Yaskawa INFORM job: R1_W49-52-A1(90,180)KM-OK.JBI

/JOB
//NAME R1_W49-52-A1(90,180)KM-OK
///FOLDERNAME KRIS-SCIANA
//POS
///NPOS 81,81,0,5,0,0
///TOOL 0
///POSTYPE PULSE
///PULSE
C00000=-7587,-78695,-93296,1458,74884,57665
C00001=105558,-78695,-93296,1458,74884,57665
C00002=105558,-78695,-93296,1458,74884,57665
C00003=54740,-7974,-10006,12021,87689,28506
C00004=74776,32390,22089,16092,92623,17270
C00005=74867,35757,29537,16050,89859,16941
C00006=75036,36599,32361,16047,88568,16832
C00007=75036,36895,33395,16047,88102,16772
C00008=74903,37254,32698,16044,88719,16805
C00009=72459,12362,8558,16008,91190,16266
C00010=61209,-17232,-1681,36622,66784,6421
C00011=61731,-16191,-908,36534,66611,6591
C00012=59990,-21702,-9204,36261,69196,6738
C00013=72720,3761,1433,15340,81732,21663
C00014=72610,7758,8804,15444,79356,21325
C00015=73045,10828,13692,15468,77892,21294
C00016=73045,11312,15266,15506,77198,21205
C00017=73045,10828,13692,15468,77892,21294
C00018=73056,12709,16349,15503,77245,21214
C00019=72823,14370,17858,15529,77218,21128
C00020=73056,12283,14967,15470,77854,21292
C00021=79642,10121,9779,4752,79820,25647
C00022=80358,6534,2777,4651,82236,25983
C00023=69953,-20577,-2415,29105,71989,-2082
C00024=71388,-15105,4995,29275,69960,-2047
C00025=71943,-12839,8075,29360,69127,-2048
C00026=71949,-11985,10076,29503,68430,-2234
C00027=71943,-12839,8075,29360,69127,-2048
C00028=78156,-21778,1298,21120,59983,2481
C00029=78744,-20042,2543,20963,59953,2712
C00030=78156,-21778,1298,21120,59983,2481
C00031=77865,-24315,-1842,21059,60645,2495
C00032=77104,-30529,-9436,20946,62223,2499
C00033=66753,-24791,-5212,33273,69818,-4262
C00034=68453,-19258,1867,33429,67885,-4157
C00035=68354,-14056,6987,33541,67521,-4315
C00036=68354,-13519,8242,33651,67105,-4449
C00037=68354,-12784,9926,33801,66552,-4629
C00038=68354,-12923,9607,33773,66657,-4594
C00039=69108,-16977,4805,33509,67096,-4131
C00040=78682,-30038,-3543,25118,55124,1302
C00041=79303,-28327,-2398,24897,55100,1566
C00042=78682,-30038,-3543,25118,55124,1302
C00043=75986,-28450,-4438,25449,57169,654
C00044=75599,-31023,-7408,25413,57744,634
C00045=74583,-37366,-14608,25368,59113,542
C00046=54832,-34796,3895,72693,39731,39244
C00047=56965,-32089,5608,72268,38461,39820
C00048=57588,-30877,10011,80435,36175,35219
C00049=57943,-31847,4343,71137,38137,40613
C00050=56828,-32279,5486,72299,38543,39782
C00051=56257,-29828,13363,87123,37301,31673
C00052=56951,-32108,5596,72272,38470,39816
C00053=54817,-34814,3883,72695,39739,39240
C00054=70512,18761,16215,24928,63616,33333
C00055=71552,23284,21050,24721,62713,33555
C00056=71200,18616,16875,24804,62971,33467
C00057=70825,17807,14425,24705,64080,33568
C00058=67755,12532,11412,25844,64241,32344
C00059=67541,9161,7476,25769,64930,32423
C00060=66799,6994,5573,25983,65214,32188
C00061=71450,3986,10861,16686,71001,58886
C00062=83506,38901,46150,14860,73867,63488
C00063=83544,40808,50439,14978,72254,63301
C00064=72489,19688,28494,17099,68495,-19316
C00065=72729,20279,28486,17025,68740,-19190
C00066=86246,35765,44483,7660,69456,64556
C00067=83439,39894,48722,4111,67251,63742
C00068=81920,28066,37949,6469,61442,62824
C00069=80051,2111,23117,10924,39735,59719
C00070=82415,-8846,23843,4944,20359,59825
C00071=68873,-12309,21104,25070,22681,48537
C00072=68288,-12793,20764,25848,22814,48089
C00073=68024,-12940,20839,26306,22782,47835
C00074=67958,-13479,20947,26756,22492,47608
C00075=67911,-23908,2369,21552,28082,50172
C00076=67911,-23908,2369,21552,28082,50172
C00077=73405,-104993,-53637,20388,20000,51360
C00078=27978,-168994,-134866,21563,-5876,50681
C00079=117827,-168994,-134866,21563,-5876,50681
C00080=64827,-168994,-134866,21563,-5876,50681
BC00000=61902,753087,991662
BC00001=7382,751982,991662
BC00002=7382,1232959,991662
BC00003=41401,1216769,518914
BC00004=54510,1210531,336745
BC00005=54510,1189341,336745
BC00006=54510,1189341,336745
BC00007=54510,1189341,336745
BC00008=54510,1189341,336745
BC00009=54510,1189341,336745
BC00010=54510,1189341,336745
BC00011=54510,1189341,336745
BC00012=54510,1189341,336745
BC00013=82383,1191142,368989
BC00014=82383,1191142,368989
BC00015=82383,1191142,368989
BC00016=82383,1191142,368989
BC00017=82383,1191142,368989
BC00018=82383,1191142,368989
BC00019=82383,1191142,368989
BC00020=82383,1191142,368989
BC00021=82383,1191142,368989
BC00022=82383,1191142,368989
BC00023=120081,1191142,413938
BC00024=120081,1191142,413938
BC00025=120081,1191142,413938
BC00026=120081,1191142,413938
BC00027=120081,1191142,413938
BC00028=120081,1191142,413938
BC00029=120081,1191142,413938
BC00030=120081,1191142,413938
BC00031=120081,1191142,413938
BC00032=120081,1191142,413938
BC00033=92240,1191142,398030
BC00034=92240,1191142,398030
BC00035=92240,1191142,398030
BC00036=92240,1191142,398030
BC00037=92240,1191142,398030
BC00038=92240,1191142,398030
BC00039=92240,1191142,398030
BC00040=92240,1191142,398030
BC00041=92240,1191142,398030
BC00042=92240,1191142,398030
BC00043=92240,1191142,398030
BC00044=92240,1191142,398030
BC00045=92240,1191142,398030
BC00046=53400,1191142,369839
BC00047=54054,1191142,349350
BC00048=54316,1191142,341155
BC00049=54316,1191142,341155
BC00050=54316,1191142,341155
BC00051=86854,1191142,340272
BC00052=86592,1191142,348467
BC00053=85937,1191142,368955
BC00054=29761,1191142,318980
BC00055=30700,1191142,309584
BC00056=30700,1191142,309584
BC00057=30700,1191142,309584
BC00058=37841,1191142,292738
BC00059=36902,1191142,302135
BC00060=34556,1191142,325626
BC00061=58988,1191142,416009
BC00062=58988,1191142,416009
BC00063=58988,1191142,416009
BC00064=57963,1191142,388162
BC00065=57963,1191142,388162
BC00066=58988,1191142,416009
BC00067=58988,1191142,416009
BC00068=58988,1191142,416009
BC00069=58988,1191142,416009
BC00070=58988,1191142,416008
BC00071=58988,1191142,416008
BC00072=58988,1191142,416008
BC00073=58988,1191142,416008
BC00074=58988,1191142,416008
BC00075=58988,1191142,416008
BC00076=58988,1191142,416008
BC00077=58988,1191142,416008
BC00078=8928,1190598,1065226
BC00079=8928,1190598,1065226
BC00080=8928,698634,1065226
///POSTYPE BASE
///RECTAN
///RCONF 0,0,0,0,0,0,0,0,0,0,0,0,0,0,0,0,0,0,0,0,0,0,0,0
P00006=0.222,-3.123,-1.508,0.0000,0.0000,0.0000
P00023=0.143,-0.036,0.682,0.0000,0.0000,0.0000
P00024=0.145,-0.552,1.326,0.0000,0.0000,0.0000
P00026=0.562,-0.002,-0.337,0.0000,0.0000,0.0000
P00027=-0.746,0.015,-9.096,0.0000,0.0000,0.0000
//INST
///DATE 2024/07/25 10:26
///ATTR SC,RW
///GROUP1 RB1,BS1
NOP
'r1_W49-52-A1(90,180)
SFTOF
MOVJ C00000 BC00000 VJ=80.00
MOVJ C00001 BC00001 VJ=80.00
MOVJ C00002 BC00002 VJ=80.00
MOVJ C00003 BC00003 VJ=100.00
MOVJ C00004 BC00004 VJ=50.00
MOVJ C00005 BC00005 VJ=20.00
MOVL C00006 BC00006 V=60.0
REFP 3 C00007 BC00007
CALL JOB:SEARCH-R1
SET P026 P006
SFTON P026
MOVL C00008 BC00008 V=60.0
MOVL C00009 BC00009 V=100.0
MOVL C00010 BC00010 V=83.3
REFP 3 C00011 BC00011
CALL JOB:SEARCH-R1
SET P026 P006
SFTON P026
MOVL C00012 BC00012 V=60.0
'Path S1206
SFTOF
MOVJ C00013 BC00013 VJ=50.00
MOVJ C00014 BC00014 VJ=50.00
MOVL C00015 BC00015 V=60.0
REFP 3 C00016 BC00016
CALL JOB:SEARCH-R1
SET P024 P006
SFTON P024
MOVL C00017 BC00017 V=100.0
MOVL C00018 BC00018 V=60.0
REFP 3 C00019 BC00019
CALL JOB:SEARCH-R1
SET P024 P006
SFTON P024
MOVL C00020 BC00020 V=60.0
MOVL C00021 BC00021 V=100.0
MOVL C00022 BC00022 V=166.7
'Path S1207
SFTOF
MOVJ C00023 BC00023 VJ=50.00
MOVJ C00024 BC00024 VJ=50.00
MOVL C00025 BC00025 V=133.3
REFP 3 C00026 BC00026
CALL JOB:SEARCH-R1
SET P023 P006
SFTON P023
MOVL C00027 BC00027 V=60.0
MOVL C00028 BC00028 V=60.0
REFP 3 C00029 BC00029
CALL JOB:SEARCH-R1
SET P023 P006
SFTON P023
MOVL C00030 BC00030 V=60.0
MOVL C00031 BC00031 V=100.0
MOVL C00032 BC00032 V=100.0
'Path S1208
SFTOF
MOVJ C00033 BC00033 VJ=50.00
MOVJ C00034 BC00034 VJ=50.00
MOVL C00035 BC00035 V=100.0
MOVL C00036 BC00036 V=100.0
REFP 3 C00037 BC00037
CALL JOB:SEARCH-R1
SET P027 P006
SFTON P027
MOVL C00038 BC00038 V=166.7
MOVL C00039 BC00039 V=166.7
MOVL C00040 BC00040 V=166.7
REFP 3 C00041 BC00041
CALL JOB:SEARCH-R1
SET P027 P006
SFTON P027
MOVL C00042 BC00042 V=60.0
MOVL C00043 BC00043 V=100.0
MOVL C00044 BC00044 V=100.0
MOVL C00045 BC00045 V=166.7
'Path W1209
SFTOF
SFTON P027
MOVJ C00046 BC00046 VJ=20.00
MOVJ C00047 BC00047 VJ=20.00
MOVL C00048 BC00048 V=166.7 PL=0
REFP 1 C00049 BC00049
REFP 2 C00050 BC00050
MACRO1 MJ#(0) ARGF7
SFTON P023
ARCON
MOVL C00051 BC00051 V=7.5
ARCOF
MOVL C00052 BC00052 V=166.7
MOVL C00053 BC00053 V=166.7
SFTOF
'Path W1210
SFTOF
SFTON P024
MOVJ C00054 BC00054 VJ=20.00
MOVL C00055 BC00055 V=100.0 PL=0
REFP 1 C00056 BC00056
REFP 2 C00057 BC00057
MACRO1 MJ#(0) ARGF6
ARCON
WVON WEV#(40)
MOVL C00058 BC00058 V=7.5
ARCOF
WVOF
MOVL C00059 BC00059 V=166.7
MOVL C00060 BC00060 V=166.7
SFTOF
'Path W1212
SFTOF
SFTON P026
MOVJ C00061 BC00061 VJ=20.00
MOVJ C00062 BC00062 VJ=20.00
MOVL C00063 BC00063 V=166.7 PL=0
REFP 1 C00064 BC00064
REFP 2 C00065 BC00065
MACRO1 MJ#(0) ARGF9
ARCON
MOVL C00066 BC00066 V=10.0
MOVL C00067 BC00067 V=10.0
MOVL C00068 BC00068 V=10.8
SFTON P024
MOVL C00069 BC00069 V=10.8
ARCON
MOVL C00070 BC00070 V=10.8
MOVL C00071 BC00071 V=10.3
MOVL C00072 BC00072 V=10.3
MOVL C00073 BC00073 V=10.3
MOVL C00074 BC00074 V=10.3
ARCOF
MOVL C00075 BC00075 V=166.7
MOVL C00076 BC00076 V=166.7
SFTOF
MOVJ C00077 BC00077 VJ=100.00
MOVJ C00078 BC00078 VJ=100.00
MOVJ C00079 BC00079 VJ=100.00
MOVJ C00080 BC00080 VJ=100.00
END
